// TIA Portal V20 export
TYPE "LKinCtrl_PathEditor_typeKinUnitTextList"
// stored: Access Published
   STRUCT
      length { ExternalAccessible := 'False'; ExternalVisible := 'False'; ExternalWritable := 'False'} : WString[7];
      angle { ExternalAccessible := 'False'; ExternalVisible := 'False'; ExternalWritable := 'False'} : WString[7];
      lengthVelocity { ExternalAccessible := 'False'; ExternalVisible := 'False'; ExternalWritable := 'False'} : WString[7];
      angleVelocity { ExternalAccessible := 'False'; ExternalVisible := 'False'; ExternalWritable := 'False'} : WString[7];
   END_STRUCT;
END_TYPE
